{attribute 'qualified_only'}
VAR_GLOBAL
	//Temperature input from EL3214 Channel1
	iiAnalogueIn_1 AT%IB100: INT;
	
	//Analogue outputs EL4002
	iqAnalogueOut_1 AT%QB100: INT;
	iqAnalogueOut_2 AT%QB102: INT;
	
END_VAR

(* stored: Version 1.1.0.1, ProductVersion 3.1.4022.10
   GVL Global_IO: Id {2a5675cd-f9a5-4b29-8d57-a071f0a61152} *)
